{attribute 'GeneratedUsingTerminal: EL3773-0000-0021'}
{attribute addProperty BoxType "EL3773-0000-0021"}
{attribute addProperty Id "LowUDINT4HiUDINT4"}
{attribute addProperty CRC "48284104"}
{attribute addProperty Size "8"}
TYPE StartTimeNextLatch_02E0C1C8 :
STRUCT
	{attribute addProperty Name "Low"}
	Low : UDINT;
	{attribute addProperty Name "Hi"}
	Hi : UDINT;
END_STRUCT
END_TYPE

(* stored: Version 1.2.0.0, ProductVersion 3.1.4024.11
   DUT StartTimeNextLatch_02E0C1C8: Id {08999750-860d-0fd4-3dc6-17574dbb80f2} *)
